FUNCTION_BLOCK MASTER

VAR_INPUT
	START  : BOOL;
	STOP   : BOOL;
	EMERG  : BOOL;
	ACK    : BOOL;
END_VAR

VAR_OUTPUT
	H1         : BOOL;
	H2         : BOOL;
	H3     	   : BOOL;
	RIPRISTINO : BOOL;
END_VAR

VAR
END_VAR

VAR_STAT
	enable      : BOOL := FALSE;
	emergenza   : BOOL := FALSE;
	acknowledge : BOOL := FALSE;
END_VAR

IF(EMERG = FALSE) THEN
	enable := FALSE;
	emergenza := TRUE;
	H2 := TRUE;
	
ELSIF(emergenza = TRUE AND ACK = TRUE) THEN
	emergenza := FALSE;
	H2 := FALSE;
	H3 := TRUE;
	acknowledge := TRUE;
	
END_IF

IF(acknowledge = TRUE
	AND ZONE.Z1.libero = TRUE
	AND ZONE.Z2.libero = TRUE
	AND ZONE.Z3.libero = TRUE
	AND ZONE.Z4.libero = TRUE
	AND ZONE.Z5.libero = TRUE
	AND ZONE.Z6.libero = TRUE) THEN
	
	acknowledge := FALSE;
	H3 := FALSE;
	H1 := FALSE;
END_IF

END_FUNCTION_BLOCK

(* stored: Version 1.1.0.1, ProductVersion 3.1.4024.12
   POU MASTER: Id {4cd99944-6bec-4dae-97df-6d0dac773983}, SpecialFunc None *)
